TYPE ParIDAccess_monitor_typ :
STRUCT
END_STRUCT
END_TYPE

(* stored: Version 1.1.0.1, ProductVersion 3.1.4024.3
   DUT ParIDAccess_monitor_typ: Id {9618d40d-0de5-043b-3aa9-d0970e7d6090} *)
